Staubli VAL3: CircleCenter.pjx

--- CircleCenter.pjx ---
Parameters version=s7.3 stackSize=5000 millimeterUnit=true
Program file=CheckMode.pgx
Program file=Circle3point.pgx
Program file=ComThOffset.pgx
Program file=MainPage.pgx
Program file=Move.pgx
Program file=OnStart.pgx
Program file=ShowOffset.pgx
Program file=init.pgx
Program file=leftPos.pgx
Program file=list.pgx
Program file=readme.pgx
Program file=start.pgx
Program file=stop.pgx
Data file=CircleCenter.dtx
Library alias=user path=Disk://userPage/userPage.pjx autoload=true password=
Library alias=MotionPage path=./MotionPage/MotionPage.pjx autoload=true password=
Library alias=date path=Disk://dateBase/dateBase.pjx autoload=true password=

--- CircleCenter.dtx ---
bool bExit
public bool bFrameSave
bool bFrameTeach
bool bOk
bool bSame = true
frame fFrame1 = {fatherId=world[0]}
frame fFrameRef = {fatherId=world[0]}
mdesc mNomSpeed
num nAngle
num nDia
num nFrame1Err = -1
num nItem[6]
num nMax[6]
num nMin[6]
num nSelectedPt = 2
num nStatus = 2
num nWorkingMode = 3
public pointRx pFrameRefPt[3]
  [0] = {x=250, z=1944, shoulder=lefty, elbow=epositive, wrist=wpositive, fatherId=world[0]}
  [1] = {x=250, z=1944, shoulder=lefty, elbow=epositive, wrist=wpositive, fatherId=world[0]}
  [2] = {x=250, z=1944, shoulder=lefty, elbow=epositive, wrist=wpositive, fatherId=world[0]}
pointRx pPointCenter = {fatherId=world[0]}
string sButton[2]
  [0] = "是"
  [1] = "否"
string sCutPosStatus
string sEmptyOrNotC[3]
string sItem[6]
string sOffSet[6]
  [0] = "X:  1460.6 "
  [1] = "Y:  35.71"
  [2] = "Z:  -199.19"
  [3] = "Rx: -0.12"
  [4] = "Ry: -0.31"
  [5] = "Rz: -53.75"
string sThreeOffset[3]
  [0] = "第1点(圆周上)"
  [1] = "第2点(圆周上)"
  [2] = "第3点(圆周上)"
tool tTool = {fatherId=flange[0], ioLink=valve1}
trsf trFrame
trsf trOffSetOut
trsf trOffset

--- CheckMode.pgx ---
program CheckMode()
begin
  while !bExit
    nWorkingMode=workingMode(nStatus)
    if nWorkingMode==1
      if nStatus!=0
        resetMotion()
        if taskStatus("Move")==150
          taskResume("Move",1)
          resetMotion()
        endIf
      endIf
    else
      resetMotion()
    endIf
    delay(0)
  endWhile
  resetMotion()
end

--- ComThOffset.pgx ---
program ComThOffset()
begin
  //-----------------------------------------------------------------------
  //Header begin
  //Description of program
  //  计算坐标系值
  //Input parameters
  //
  //Output paramaters
  //
  //Example
  //  call ComputeThOffset()
  //History
  //  Creation : 2012-06-11 - PF.Zhong
  //Header end
  //-----------------------------------------------------------------------

  nFrame1Err=setFrame(pFrameRefPt[0],pFrameRefPt[1],pFrameRefPt[2],fFrame1)
  if nFrame1Err==-1
    popUpMsg("X方向点离原点太近")
  endIf
  if nFrame1Err==-2
    popUpMsg("Y方向点离原点太近")
  endIf
  if nFrame1Err==0
    trOffset=fFrame1.trsf
  else
  endIf
end

--- list.pgx ---
program list(string pTitle (dimensions=1), num pX (dimensions=1), num pY (dimensions=1), num pDx (dimensions=1), num pDy (dimensions=1), string& sName[] (dimensions=1))
  local num lDx
  local num lDy
  local num lI
  local num lJ
  local string lStr
  local string lStrLine
  local num lValue
  local num l_nsize
begin
  //-----------------------------------------------------------------------
  //Header begin
  //Description of program
  //  在列pX和行pY处创建宽pDx，高pDy的列表；列表名称pTitle；列表内容为sName
  //Input parameters
  //  string pTitle:列表名
  //  num pX: 列表左上角列位置
  //  num PY: 列表左上角行位置
  //  num pDx: 列表宽
  //  num pDy：列表高
  //  string sName:列表显示内容
  //Output paramaters
  //
  //Example
  //  call list("list1",10,0,20,20)
  //Creation : 2012-06-11 - PF.Zhong
  //Header end
  //-----------------------------------------------------------------------
  //
  lStrLine="─────────────────────────────────────────"
  lDx=pDx
  lDy=pDy
  l_nsize=size(sName)
  //Top
  lStr="┌"+mid(lStrLine,lDx,0)+"┐"
  gotoxy(pX,pY)
  put(lStr)
  lValue=pX+2
  //Title
  if pTitle!=""
    call leftPos("┤"+pTitle+"├",lDx,pTitle)
    gotoxy(pX+lDx-getDisplayLen(pTitle)+1,pY)
    put(pTitle)
  endIf
  //Containt
  for lJ=1 to lDy
    lValue=pY+lJ
    lStr="│"
    gotoxy(pX,lValue)
    put(lStr)
    if lJ<=l_nsize
      if sName[lJ-1]!=""
        put(sName[lJ-1])
      endIf
    endIf
    gotoxy(pX+lDx+1,lValue)
    put(lStr)
  endFor
  //Bottom
  lValue=pY+lJ
  lStr="└"+mid(lStrLine,lDx,0)+"┘"
  gotoxy(pX,lValue)
  put(lStr)
end

--- OnStart.pgx ---
public program OnStart(tool& x_tTool, trsf& x_trFrameOut)
begin
  //-----------------------------------------------------------------------
  //Header begin
  //Description of program
  //
  //Input parameters
  //  tool x_tTool:工具
  //  frame x_fFrame:参考坐标系

  //Output paramaters
  //  trsf x_trOffSetOut:新建坐标系的trsf值
  //
  //Example
  //  call OnStart(tool,frame,trTrsfSetOut)
  //History
  //  Creation : 2012-06-11 - PF.Zhong
  //Header end
  //-----------------------------------------------------------------------
  call init(x_tTool)
  if taskStatus("CheckModeFrame")!=-1
    taskKill("CheckModeFrame")
    wait(taskStatus("CheckModeFrame")==-1)
  endIf
  taskCreate "CheckModeFrame",15,CheckMode()
  call MainPage(x_trFrameOut)
end

--- readme.pgx ---
program readme()
begin
  //Title:示教坐标系

  //General description:
  //通过三点示教坐标系；

  //Hardware required:

  //Val3 Option:
  //Val3 version：s7.1以上；
  //Val3 license:
  //Val3 addon：对应val3版本的addon--expansion、motion、recorder、relbo、remote和velocity

  //Variables:
  //bool:
  //  bAlignDone:对齐是否完成标识符
  //  bFrameSave:坐标系示教是否完成标识符
  //  bPC:是否与上位机通讯标识符
  //  bSame:字符串是否变化标识符

  //frame
  //  frame1:坐标系

  //mdesc
  //  mNomSpeed:默认速度

  //num
  //  nFrame1Err:建立坐标系返回值
  //  nItem[6]:储存point类型的6个位置分量
  //  nMax[6]:输入最大值
  //  nMin[6]:输入最小
  //  nSelectedPt:选择点编号
  //

  //point
  //  pFrameRefPt[3]:构成frame的三个点

  //string:
  //  sCutPosStatus:字符串标志符
  //  sEmptyOrNotC:字符串标志符
  //  sItem[6]:point的6个分量的字符串形式
  //  sOffSet[6]:frame的6个分量的字符串形式
  //  sThreeOffset[3]:构成frame的三个点的字符串形式


  //tool
  //  tTool:工具

  //trsf
  //  trOffset:frame的trsf值
  //  trOffsetOut:frame的trsf值的输出变量



  //Included libraries:
  //DataBase：与PC交换的公共数据和其他库共同使用的数据
  //PublicProg:公共函数库
  //userPage：通用界面函数库

  //Miscellaneous：

  //Keywords:

  //other:
end
